RoboDK station: test1.rdk

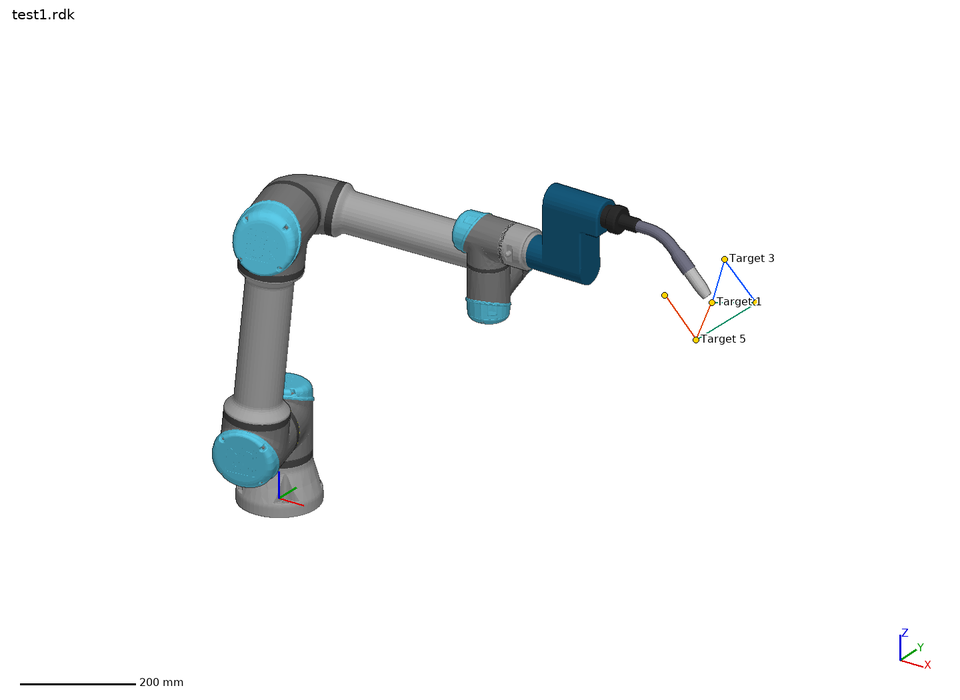
[picture v0: the station drawn from its stored meshes, robots at their saved joint values, targets as dots, program paths as lines]
Station test1 (saved by RoboDK 5.2.2). Poses are relative to the parent item; angles as X-Y-Z fixed-axis rotations.
  - frame UR5e Base at (0, 0, 0) mm
    - robot UR5e: 6 axes, payload 5 kg, reach 850 mm, repeatability 0.03 mm, weight 18.4 kg
        modified DH rows (alpha deg, a mm, theta deg, d mm): 0, 0, 0, 162.5; 90, 0, 180, 0; 0, 425, 0, 0; 0, 392.25, 0, 133.3; -90, 0, 0, 99.7; 90, 0, 180, 99.6
        joint limits [-360, -360, -360, -360, -360, -360] to [360, 360, 360, 360, 360, 360]; home [0, -90, -90, 0, 90, 0]; saved at [16.021, -95.182, -92.617, 7.799, 73.979, 90]
      - tool Weld gun, TCP at (-4, 0, 371.3) mm, rotated rx 0 ry 45 rz 0 deg, size 299.9 x 60 x 318.3 mm
    - target Target 1 (Cartesian target) at (918.11, -10.27, 636.24) mm, rotated rx -180 ry 45 rz -180 deg; joints [16.021, -95.182, -92.617, 7.799, 73.979, 90] of UR5e
    - target Target 2 (Cartesian target) at (947, 81.88, 607.35) mm, rotated rx -180 ry 45 rz -180 deg; joints [25.776, -100.793, -90.429, 11.222, 64.224, 90] of UR5e
    - target Target 3 (Cartesian target) at (881.44, 80.08, 672.91) mm, rotated rx -180 ry 45 rz -180 deg; joints [29.621, -90.626, -92.043, 2.669, 60.379, 90] of UR5e
    - target Target 4 (Cartesian target) at (879.65, -96.59, 674.7) mm, rotated rx -180 ry 45 rz -180 deg; joints [5.209, -90.861, -91.543, 2.404, 84.791, 90] of UR5e
    - target Target 5 (Cartesian target) at (946.41, -97.59, 607.94) mm, rotated rx -180 ry 45 rz -180 deg; joints [4.341, -101.097, -89.972, 11.069, 85.659, 90] of UR5e
  - program Prog1 (6 instructions, listed below)
  - program Prog2 (6 instructions, listed below)
  - program Prog3 (6 instructions, listed below)
  - Python program Prog2 (listed below)
  - Python program SampleOfflineProgramming (listed below)
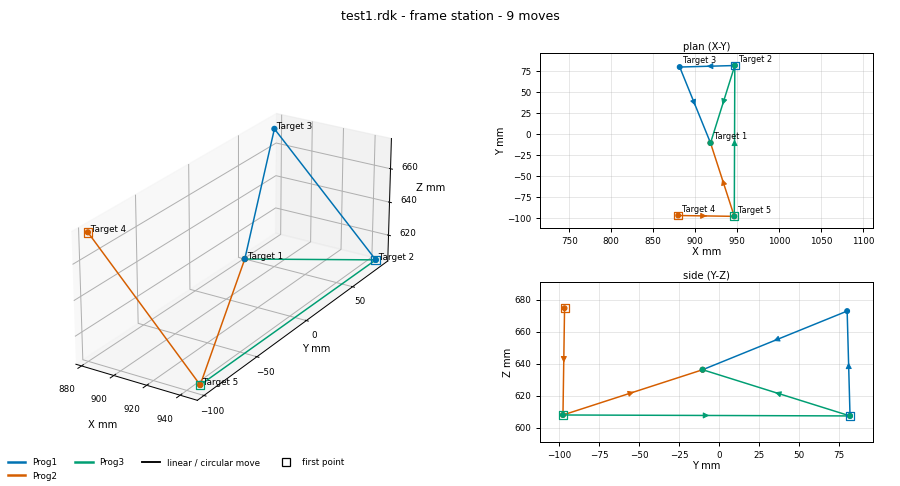
[picture p0: tool path of test1.rdk in frame station, 9 of 9 moves have a stored position in this frame; points joined in program order, loops and branches not executed]

--- program Prog1 (robot UR5e) ---
  Set speed (50.0 mm/s)
  Set Ref.: UR5e Base
  Set Tool: Weld gun
  MoveL (Target 2)
  MoveL (Target 3)
  MoveL (Target 1)

--- program Prog2 (robot UR5e) ---
  Set speed (50.0 mm/s)
  Set Ref.: UR5e Base
  Set Tool: Weld gun
  MoveL (Target 4)
  MoveL (Target 5)
  MoveL (Target 1)

--- program Prog3 (robot UR5e) ---
  Set speed (50.0 mm/s)
  Set Ref.: UR5e Base
  Set Tool: Weld gun
  MoveL (Target 5)
  MoveL (Target 2)
  MoveL (Target 1)

--- Python program Prog2 ---
from robolink import *
from robodk import *

import PySimpleGUI as sg
import os.path

sg.theme('DarkBlack')

bottomCoverColor = 0
fuseAmount = 0
topCoverType = 0
topCoverColor = 0
engraving = "No text"

selectColor = (
    'Black', 'White', 'Blue')

selectFuse = (
    '0', '1', '2')

selectTopCoverType = (
    'Flat', 'Curved')

width = max(map(len, selectColor))+1

layout = [
    [sg.Text("Select bottom cover color")], [sg.Combo(selectColor, size=(width, 5), enable_events=True, key='SBCC')],
    [sg.Text("Select amount of fuses")], [sg.Combo(selectFuse, size=(width, 5), enable_events=True, key='SAOF')],
    [sg.Text("Select top cover type")], [sg.Combo(selectTopCoverType, size=(width, 5), enable_events=True, key='STCT')],
    [sg.Text("Select top cover color")], [sg.Combo(selectColor, size=(width, 5), enable_events=True, key='STCC')],
    [sg.Text("Choose engraving")], [sg.Input(do_not_clear=True, enable_events=True, key='textbox')],
    [sg.Button("Place order", key='PO')],
]

window = sg.Window("Dummy Phone Order", layout, finalize=True)

while True:
    event, values = window.read()
    print(event, values)

    #Textbox
    if len(values["textbox"])>10:
        window.Element('textbox').Update(values['textbox'][:-1])

    #Bottom cover color
    if values['SBCC'] == "Black":
        bottomCoverColor = 1

    if values['SBCC'] == "White":
        bottomCoverColor = 2

    if values['SBCC'] == "Blue":
        bottomCoverColor = 3

    #Fuse amount
    if values['SAOF'] == "0":
        fuseAmount = 1

    if values['SAOF'] == "1":
        fuseAmount = 2

    if values['SAOF'] == "2":
        fuseAmount = 3

    #Top cover type
    if values['STCT'] == "Flat":
        topCoverType = 1

    if values['STCT'] == "Curved":
        topCoverType = 2

    #Top cover color
    if values['STCC'] == "Black":
        topCoverColor = 1

    if values['STCC'] == "White":
        topCoverColor = 2

    if values['STCC'] == "Blue":
        topCoverColor = 3

    if event == sg.WINDOW_CLOSED:
        break

    if event == 'PO':
        if bottomCoverColor == 0 or fuseAmount == 0 or topCoverType == 0 or topCoverColor == 0:
            sg.popup_error(f'Fill everything out!')
        else:
            #Place order
            break

window.close()

print(bottomCoverColor, fuseAmount, topCoverType, topCoverColor)

RL = Robolink()

robot = RL.Item('UR5e')

home = RL.Item('Target 1')

if bottomCoverColor == 1:
    assemble1 = RL.Item('Prog1')
    assemble1.RunProgram()

if bottomCoverColor == 2:
    assemble2 = RL.Item('Prog3')
    assemble2.RunProgram()

--- Python program SampleOfflineProgramming ---
# This macro shows an example to draw a polygon of radius R and n_sides vertices using the RoboDK API for Python
# More information about the RoboDK API here:
# https://robodk.com/doc/en/RoboDK-API.html
from robolink import *    # API to communicate with RoboDK
from robodk import *      # robodk robotics toolbox

# Any interaction with RoboDK must be done through RDK:
RDK = Robolink()

# Select a robot (popup is displayed if more than one robot is available)
robot = RDK.ItemUserPick('Select a robot', ITEM_TYPE_ROBOT)
if not robot.Valid():
    raise Exception('No robot selected or available')


# get the current position of the TCP with respect to the reference frame:
# (4x4 matrix representing position and orientation)
target_ref = robot.Pose()
pos_ref = target_ref.Pos()
print("Drawing a polygon around the target: ")
print(Pose_2_TxyzRxyz(target_ref))


# move the robot to the first point:
robot.MoveJ(target_ref)

# It is important to provide the reference frame and the tool frames when generating programs offline
robot.setPoseFrame(robot.PoseFrame())
robot.setPoseTool(robot.PoseTool())
robot.setZoneData(10) # Set the rounding parameter (Also known as: CNT, APO/C_DIS, ZoneData, Blending radius, cornering, ...)
robot.setSpeed(200) # Set linear speed in mm/s

# Set the number of sides of the polygon:
n_sides = 6
R = 100

# make a hexagon around reference target:
for i in range(n_sides+1):
    ang = i*2*pi/n_sides #angle: 0, 60, 120, ...

    #-----------------------------
    # Movement relative to the reference frame
    # Create a copy of the target
    target_i = Mat(target_ref)
    pos_i = target_i.Pos()
    pos_i[0] = pos_i[0] + R*cos(ang)
    pos_i[1] = pos_i[1] + R*sin(ang)
    target_i.setPos(pos_i)
    print("Moving to target %i: angle %.1f" % (i, ang*180/pi))
    print(str(Pose_2_TxyzRxyz(target_i)))
    robot.MoveL(target_i)

    #-----------------------------
    # Post multiply: relative to the tool
    #target_i = target_ref * rotz(ang) * transl(R,0,0) * rotz(-ang)
    #robot.MoveL(target_i)

# move back to the center, then home:
robot.MoveL(target_ref)

print('Done')
